// TwinCAT 3 PLC project LabExercise
// ProgramVersion: 3.1.4023.0
// libraries:
//   Tc2_NCI, * (Beckhoff Automation GmbH)
//   Tc2_Standard, * (Beckhoff Automation GmbH)
//   Tc2_System, * (Beckhoff Automation GmbH)
//   Tc3_Module, * (Beckhoff Automation GmbH)
//   VisuDialogs, * (System)
// project tree:
//   Comissioning/Function blocks/ FB_ModifyAutomaticControlSettings.TcPOU (not stored)
//   Comissioning/GVLs/ G_Commissioning.TcGVL (not stored)
//   Comissioning/Struct/ ST_AutomaticControlSettings.TcDUT (not stored), ST_ClosedLoopControlSettings.TcDUT (not stored), ST_MotionReferenceGeneratorSettings.TcDUT (not stored), ST_OpenLoopControlSettings.TcDUT (not stored)
//   ControlBox/Interfaces/ I_ControlBox.TcIO
//   ControlBox/Function blocks/ FB_ControlBox.TcPOU, FB_RealControlBox.TcPOU, FB_VirtualControlBox.TcPOU
//   CraneControl/Function blocks/Sub blocks/ FB_ActiveDamping.TcPOU, FB_Clock.TcPOU, FB_ClosedLoopControl.TcPOU, FB_Joystick.TcPOU, FB_MotionReferenceGenerator_limit.TcPOU, FB_OpenLoopControl.TcPOU, FB_ResetIntegralController.TcPOU, FB_Status.TcPOU
//   CraneControl/Enums/ E_Mode.TcDUT, E_Status.TcDUT
//   CraneControl/Function blocks/Main blocks/ FB_AutomaticControl.TcPOU, FB_ManualControl.TcPOU
//   CraneControl/Functions/ F_BarToEng.TcPOU (not stored), F_LminToEng.TcPOU (not stored), F_RadToDeg.TcPOU (not stored)
//   CraneControl/GVLs/ G_Parameters.TcGVL (not stored), G_Work.TcGVL
//   CraneControl/Struct/ ST_ActiveDamping.TcDUT, ST_Parameters.TcDUT
//   / GlobalTextList.TcGTLO, PlcTask.TcTTO, Simulator.TcTTO (not stored), Visualization Manager.TcVMO (not stored)
//   HMI/ HMI.TcVIS
//   HMI/Sub/ CommissioningHMI.TcVIS, VirtualControlBox.TcVIS
//   Inputs/ FB_JoystickInputScaling.TcPOU, FB_PositionInputScaling.TcPOU, FB_PressureInputScaling.TcPOU, G_Inputs.TcGVL, G_Sensors.TcGVL
//   Inputs/Struct/ ST_AnalogInput.TcDUT (not stored), ST_AnalogInputStatus.TcDUT (not stored)
//   Outputs/ FB_ValveOutput.TcPOU, G_Outputs.TcGVL
//   Outputs/Struct/ ST_pValveDeadBand.TcDUT, ST_ValveOutput.TcDUT
//   ControlBox/GVLs/ G_VirtualControlBox.TcGVL (not stored)
//   Programs/ MAIN.TcPOU, P_Commissioning.TcPOU (not stored), P_ControlBox.TcPOU, P_CraneControl.TcPOU, P_Inputs.TcPOU, P_Outputs.TcPOU, P_Simulator.TcPOU
//   Simulator/ FB_CraneSimulator.TcPOU (not stored), G_Simulator.TcGVL
// real-time tasks:
//   TASK PlcTask: cycle T#1ms, priority 20, ADS port 350
//   TASK Simulator: cycle T#100us, priority 1, ADS port 351
// I/O:
//   DEVICE PLC (EtherCAT), AmsNetId 128.39.203.30.2.1
//     PLC Rack (EK1200) [EK1200-5000 EtherCAT Power supply (2A E-Bus)]
//       DI (EL1008) [EL1008 8Ch. Dig. Input 24V, 3ms]
//       DO (EL2008) [EL2008 8Ch. Dig. Output 24V, 0.5A]
//       End Cap 4 (EL9011) [EL9011 End Terminal]
//   DEVICE RIO (EtherCAT), AmsNetId 128.39.203.30.5.1
//     RIO (EK1100) [EK1100 EtherCAT Coupler (2A E-Bus)]
//       DI (EL1008) [EL1008 8Ch. Dig. Input 24V, 3ms]
//       DO (EL2008) [EL2008 8Ch. Dig. Output 24V, 0.5A]
//       AI1 (EL3068) [EL3068 8Ch. Ana. Input 0-10V]
//       AI2 (EL3068) [EL3068 8Ch. Ana. Input 0-10V]
//       AI3 (EL3174) [EL3174 4Ch. Ana. Input +/-10V Diff., +/-20mA SingleEnded, 16 Bit]
//       AO (EL4104) [EL4104 4Ch. Ana. Output 0-10V, 16bit]
//       End Cap (EL9011) [EL9011 End Terminal]
// variable links:
//   LabExercise/LabExercise Instance <-> PLC (EtherCAT)/PLC Rack (EK1200)/DI (EL1008)
//     PlcTask Inputs/G_Inputs.bTest <-> Channel 1/Input
//   LabExercise/LabExercise Instance <-> PLC (EtherCAT)/PLC Rack (EK1200)/DO (EL2008)
//     PlcTask Outputs/G_Outputs.bTest <-> Channel 1/Output
//   LabExercise/LabExercise Instance <-> RIO (EtherCAT)/RIO (EK1100)/AI1 (EL3068)
//     PlcTask Inputs/G_Inputs.stCylPos.nValue <-> AI Standard Channel 3/Value
//     PlcTask Inputs/G_Inputs.stCylPos.stStatus <-> AI Standard Channel 3/Status
//     PlcTask Inputs/G_Inputs.stJoyX.nValue <-> AI Standard Channel 1/Value
//     PlcTask Inputs/G_Inputs.stJoyX.stStatus <-> AI Standard Channel 1/Status
//     PlcTask Inputs/G_Inputs.stJoyY.nValue <-> AI Standard Channel 2/Value
//     PlcTask Inputs/G_Inputs.stJoyY.stStatus <-> AI Standard Channel 2/Status
//     PlcTask Inputs/G_Inputs.stSpoolPos.nValue <-> AI Standard Channel 4/Value
//     PlcTask Inputs/G_Inputs.stSpoolPos.stStatus <-> AI Standard Channel 4/Status
//   LabExercise/LabExercise Instance <-> RIO (EtherCAT)/RIO (EK1100)/AI2 (EL3068)
//     PlcTask Inputs/G_Inputs.stPressureCompensator.nValue <-> AI Standard Channel 3/Value
//     PlcTask Inputs/G_Inputs.stPressureCompensator.stStatus <-> AI Standard Channel 3/Status
//     PlcTask Inputs/G_Inputs.stPressureLhvSide.nValue <-> AI Standard Channel 5/Value
//     PlcTask Inputs/G_Inputs.stPressureLhvSide.stStatus <-> AI Standard Channel 5/Status
//     PlcTask Inputs/G_Inputs.stPressurePistonSide.nValue <-> AI Standard Channel 4/Value
//     PlcTask Inputs/G_Inputs.stPressurePistonSide.stStatus <-> AI Standard Channel 4/Status
//     PlcTask Inputs/G_Inputs.stPressureReturn.nValue <-> AI Standard Channel 2/Value
//     PlcTask Inputs/G_Inputs.stPressureReturn.stStatus <-> AI Standard Channel 2/Status
//     PlcTask Inputs/G_Inputs.stPressureRodSide.nValue <-> AI Standard Channel 6/Value
//     PlcTask Inputs/G_Inputs.stPressureRodSide.stStatus <-> AI Standard Channel 6/Status
//     PlcTask Inputs/G_Inputs.stPressureSupply.nValue <-> AI Standard Channel 1/Value
//     PlcTask Inputs/G_Inputs.stPressureSupply.stStatus <-> AI Standard Channel 1/Status
//   LabExercise/LabExercise Instance <-> RIO (EtherCAT)/RIO (EK1100)/AI3 (EL3174)
//     PlcTask Inputs/G_Inputs.stFlowReturnSide.nValue <-> AI Standard Channel 1/Value
//     PlcTask Inputs/G_Inputs.stFlowReturnSide.stStatus <-> AI Standard Channel 1/Status
//   LabExercise/LabExercise Instance <-> RIO (EtherCAT)/RIO (EK1100)/AO (EL4104)
//     PlcTask Outputs/G_Outputs.stValveOutput.nValveOutput <-> AO Output Channel 1/Analog output
//   LabExercise/LabExercise Instance <-> RIO (EtherCAT)/RIO (EK1100)/DI (EL1008)
//     PlcTask Inputs/G_Inputs.bAutoModeSelector <-> Channel 1/Input
//     PlcTask Inputs/G_Inputs.bManualModeSelector <-> Channel 2/Input
//     PlcTask Inputs/G_Inputs.bStartButton <-> Channel 3/Input
//     PlcTask Inputs/G_Inputs.bStopButton <-> Channel 4/Input
//   LabExercise/LabExercise Instance <-> RIO (EtherCAT)/RIO (EK1100)/DO (EL2008)
//     PlcTask Outputs/G_Outputs.bGreenLight <-> Channel 1/Output
//     PlcTask Outputs/G_Outputs.bRedLight <-> Channel 2/Output
//     PlcTask Outputs/G_Outputs.stValveOutput.bEnable <-> Channel 3/Output

CONFIGURATION LabExercise
    RESOURCE PLC ON TwinCAT3
        TASK PlcTask(INTERVAL := T#10ms, PRIORITY := 20);
        PROGRAM MAIN WITH PlcTask : MAIN;
    END_RESOURCE
END_CONFIGURATION

// ---- CraneControl/Enums/E_Mode.TcDUT
{attribute 'qualified_only'}
{attribute 'strict'}
TYPE E_Mode :
(
	Off,
	Manual,
	Auto
);
END_TYPE

// ---- CraneControl/Enums/E_Status.TcDUT
{attribute 'qualified_only'}
{attribute 'strict'}
TYPE E_Status :
(
	Off := 0,
	Fault,
	Ready,
	Starting,
	Running,
	Stopping,
	Checking
);
END_TYPE

// ---- CraneControl/Struct/ST_ActiveDamping.TcDUT
TYPE ST_ActiveDamping :
STRUCT
	fFlowGainInverse : LREAL := -1.7153E03;	
	fHPF_Num1 : LREAL := 9.019E-12;
	fHPF_Num2 : LREAL := -9.019E-12;
	fHPF_Den1 : LREAL := 1.0;
	fHPF_Den2 : LREAL := -0.9905;
	fVDI_Num1 : LREAL := 25;
	fVDI_Num2 : LREAL := -48.83;
	fVDI_Num3 : LREAL := 23.85;
	fVDI_Den1 : LREAL := 1;
	fVDI_Den2 : LREAL := -1.721;
	fVDI_Den3 : LREAL := 0.7408;
END_STRUCT
END_TYPE

// ---- CraneControl/Struct/ST_Parameters.TcDUT
TYPE ST_Parameters :
STRUCT
	fCyclicTime 						: LREAL := 0.001; //[s]
	fMaxVelocityLimit 					: LREAL := 0.05; //[m/s]
	stOpenLoopControlSettings 			: ST_OpenLoopControlSettings;
	stClosedLoopControlSettings 		: ST_ClosedLoopControlSettings;
	stPressureFeedback 					: ST_ActiveDamping;
	stValveDeadBand 					: ST_pValveDeadBand;
END_STRUCT
END_TYPE

// ---- Outputs/Struct/ST_pValveDeadBand.TcDUT
TYPE ST_pValveDeadBand :
STRUCT
	fPosMax	: LREAL := 29490; // Positive min value [19660..29490]
	fPosMin	: LREAL := 20889; // Positive max value [19660..29490]
	fNegMin : LREAL := 18441; // Negative max value [9830..19660]
	fNegMax	: LREAL := 9830; // Negative min value [9830..19660]
END_STRUCT
END_TYPE

// ---- Outputs/Struct/ST_ValveOutput.TcDUT
TYPE ST_ValveOutput :
STRUCT
	bEnable					AT %Q* : BOOL := 0;
	nValveOutput 			AT %Q* : INT := 19660;
END_STRUCT
END_TYPE

// ---- CraneControl/GVLs/G_Work.TcGVL
{attribute 'qualified_only'}
VAR_GLOBAL
	eMode 			: E_Mode;
	eStatus 		: E_Status;
	fJoystickY 		: LREAL;
	bFault 			: BOOL;
	bStartButton 	: BOOL;
	bStopButton 	: BOOL;
END_VAR

// ---- Inputs/G_Inputs.TcGVL
{attribute 'qualified_only'}
VAR_GLOBAL
	// PLC Rack
	// Digital Inputs
	bTest 						AT %I* : BOOL;
	
	// RIO Rack
	// Digital Inputs
	bAutoModeSelector			AT %I* : BOOL;
	bManualModeSelector			AT %I* : BOOL;
	bStartButton				AT %I* : BOOL;
	bStopButton					AT %I* : BOOL;
	
	// Analog Inputs 1
	stJoyX 						: ST_AnalogInput;
	stJoyY						: ST_AnalogInput;
	stCylPos 					: ST_AnalogInput;
	stSpoolPos 					: ST_AnalogInput;
	
	// Analog Inputs 2
	stPressureSupply 			: ST_AnalogInput;
	stPressureReturn 			: ST_AnalogInput;
	stPressureCompensator 		: ST_AnalogInput;
	stPressurePistonSide 		: ST_AnalogInput;
	stPressureLhvSide 		    : ST_AnalogInput;
	stPressureRodSide			: ST_AnalogInput;
	
	// Analog Inputs 3 (Multi)
	stFlowReturnSide			: ST_AnalogInput;
END_VAR

// ---- Inputs/G_Sensors.TcGVL
{attribute 'qualified_only'}
VAR_GLOBAL
	fJoystickY 			: LREAL;
	fPistonPosition 	: LREAL;
	fPressureSupply		: LREAL;
	fPressureReturn 	: LREAL;
	fPressurePistonSide : LREAL;
	fPressureLhvSide  	: LREAL;
	fPressureRodSide 	: LREAL;
END_VAR

// ---- Outputs/G_Outputs.TcGVL
{attribute 'qualified_only'}
VAR_GLOBAL
	// PLC Rack
	// Digital Outputs
	bTest					 AT %Q* : BOOL;
	
	// RIO Rack
	// Digital Outputs
	bGreenLight 			AT %Q* : BOOL;
	bRedLight 				AT %Q* : BOOL;
	// Analog Outputs
	stValveOutput : ST_ValveOutput;
END_VAR

// ---- Simulator/G_Simulator.TcGVL
{attribute 'qualified_only'}
VAR_GLOBAL
	bSimulatorOn : BOOL;
	fPistonSidePressure : LREAL;
	fRodSidePressure 	: LREAL;
	fPistonPosition 	: LREAL;
END_VAR

// ---- ControlBox/Interfaces/I_ControlBox.TcIO
INTERFACE I_ControlBox

METHOD Lamps 
VAR_INPUT
	bEnable : BOOL;
END_VAR
END_METHOD

METHOD ModeSelector 
VAR_INPUT
END_VAR
VAR_OUTPUT
	eMode : E_Mode;
END_VAR
END_METHOD

END_INTERFACE

// ---- Programs/MAIN.TcPOU
PROGRAM MAIN
VAR
END_VAR

P_Commissioning();
P_ControlBox();
P_CraneControl();
P_Outputs();
P_Inputs();

END_PROGRAM

// ---- Programs/P_ControlBox.TcPOU
PROGRAM P_ControlBox
VAR
	fbControlBox : FB_ControlBox; 
END_VAR

fbControlBox(
bRealControlBox := TRUE,
eStatus := G_Work.eStatus,
eMode => G_Work.eMode,
);

END_PROGRAM

// ---- ControlBox/Function blocks/FB_ControlBox.TcPOU
FUNCTION_BLOCK FB_ControlBox
VAR_INPUT
	bRealControlBox : BOOL;
	eStatus : E_Status;
END_VAR
VAR_OUTPUT
	eMode : E_Mode;
END_VAR
VAR
	fbVirtualControlBox : FB_VirtualControlBox;
	fbRealControlBox : FB_RealControlBox;
	fbSelectedControlBox : I_ControlBox := fbVirtualControlBox;
END_VAR

IF bRealControlBox THEN
	fbSelectedControlBox := fbRealControlBox;
ELSE
	fbSelectedControlBox := fbVirtualControlBox;
END_IF	
	
fbSelectedControlBox.ModeSelector(
	eMode => eMode
);

fbSelectedControlBox.PushButtons(
	eMode := eMode,
	eStatus := eStatus,
	bStart => G_Work.bStartButton,
	bStop => G_Work.bStopButton 	
);

fbSelectedControlBox.Lamps(
	eMode := eMode,
	eStatus := eStatus
);

fbSelectedControlBox.Joystick(
	eMode := eMode,
	eStatus := eStatus,
	fJoystickY => G_Work.fJoystickY
);

END_FUNCTION_BLOCK

// ---- ControlBox/Function blocks/FB_VirtualControlBox.TcPOU
FUNCTION_BLOCK FB_VirtualControlBox IMPLEMENTS I_ControlBox
VAR_INPUT
END_VAR
VAR_OUTPUT
END_VAR
VAR
END_VAR

METHOD Lamps
VAR_INPUT
	bEnable : BOOL;
END_VAR
IF bEnable THEN 
	IF G_Work.eStatus = E_Status.Running THEN
		G_VirtualControlBox.bGreenLight :=  TRUE;
	ELSE
		G_VirtualControlBox.bGreenLight :=  FALSE;
	END_IF
	
	IF G_Work.eStatus = E_Status.Fault THEN
		G_VirtualControlBox.bRedLight :=  TRUE;
	ELSE
		G_VirtualControlBox.bRedLight :=  FALSE;
	END_IF
END_IF
END_METHOD

METHOD ModeSelector 
VAR_INPUT
END_VAR
VAR_OUTPUT
	eMode : E_Mode;
END_VAR
CASE eMode OF 
	E_Mode.Off:	
		IF G_VirtualControlBox.bOnSelector AND NOT(G_VirtualControlBox.bAutoSelector) THEN	
			eMode := E_Mode.Manual;
		END_IF
		
		IF G_VirtualControlBox.bOnSelector AND G_VirtualControlBox.bAutoSelector THEN	
			eMode := E_Mode.Auto;
		END_IF

	E_Mode.Manual: 
		IF NOT(G_VirtualControlBox.bOnSelector) THEN	
			eMode := E_Mode.Off;
		END_IF
		
		IF G_VirtualControlBox.bOnSelector AND G_VirtualControlBox.bAutoSelector THEN	
			eMode := E_Mode.Auto;
		END_IF
	
	E_Mode.Auto:
		IF NOT(G_VirtualControlBox.bOnSelector) THEN	
			eMode := E_Mode.Off;
		END_IF
		
		IF G_VirtualControlBox.bOnSelector AND NOT(G_VirtualControlBox.bAutoSelector) THEN	
			eMode := E_Mode.Manual;
		END_IF	
ELSE 	
	eMode := E_Mode.Off;
END_CASE
END_METHOD

END_FUNCTION_BLOCK

// ---- ControlBox/Function blocks/FB_RealControlBox.TcPOU
FUNCTION_BLOCK FB_RealControlBox IMPLEMENTS I_ControlBox
VAR_INPUT
END_VAR
VAR_OUTPUT
END_VAR
VAR
END_VAR

METHOD Joystick
VAR_INPUT
	eMode 	: E_Mode;
	eStatus : E_Status;
END_VAR
VAR_OUTPUT
	fJoystickY : LREAL;
END_VAR
IF eMode = E_Mode.Manual AND eStatus = E_Status.Running THEN
	fJoystickY := G_Sensors.fJoystickY;
ELSE
	fJoystickY := 0.0;
END_IF
END_METHOD

METHOD Lamps 
VAR_INPUT
	eMode 	: E_Mode;
	eStatus : E_Status;
END_VAR
IF eStatus = E_Status.Running AND NOT(eMode = E_Mode.Off) THEN
	G_Outputs.bGreenLight :=  TRUE;
ELSE
	G_Outputs.bGreenLight :=  FALSE;
END_IF

IF eStatus = E_Status.Fault  AND NOT(eMode = E_Mode.Off) THEN
	G_Outputs.bRedLight :=  TRUE;
ELSE
	G_Outputs.bRedLight :=  FALSE;
END_IF
END_METHOD

METHOD ModeSelector 
VAR_INPUT
END_VAR
VAR_OUTPUT
	eMode : E_Mode;
END_VAR
CASE eMode OF 
	E_Mode.Off:	
		IF G_Inputs.bManualModeSelector AND NOT(G_Inputs.bAutoModeSelector) THEN	
			eMode := E_Mode.Manual;
		END_IF
		
		IF G_Inputs.bAutoModeSelector AND NOT(G_Inputs.bManualModeSelector) THEN	
			eMode := E_Mode.Auto;
		END_IF

	E_Mode.Manual: 
		IF NOT(G_Inputs.bManualModeSelector) AND NOT(G_Inputs.bManualModeSelector) THEN	
			eMode := E_Mode.Off;
		END_IF
		
		IF G_Inputs.bAutoModeSelector AND NOT(G_Inputs.bManualModeSelector) THEN	
			eMode := E_Mode.Auto;
		END_IF
	
	E_Mode.Auto:
		IF NOT(G_Inputs.bManualModeSelector) AND NOT(G_Inputs.bManualModeSelector) THEN	
			eMode := E_Mode.Off;
		END_IF
		
		IF G_Inputs.bManualModeSelector AND NOT(G_Inputs.bAutoModeSelector) THEN	
			eMode := E_Mode.Manual;
		END_IF	
ELSE 	
	eMode := E_Mode.Off;
END_CASE
END_METHOD

METHOD PushButtons
VAR_INPUT
	eMode 	: E_Mode;
	eStatus : E_Status;
END_VAR
VAR_OUTPUT
	bStart : BOOL;
	bStop : BOOL;
END_VAR
IF NOT(eMode = E_Mode.Off) AND (NOT(eStatus = E_Status.Fault) OR (eStatus = E_Status.Off)) THEN 
	bStart := G_Inputs.bStartButton;
	bStop := G_Inputs.bStopButton;
ELSE
	bStart := FALSE;
	bStop := FALSE;
END_IF
END_METHOD

END_FUNCTION_BLOCK

// ---- Programs/P_CraneControl.TcPOU
PROGRAM P_CraneControl
VAR
 	fbStatus 					: FB_Status;
	fbRunningClock 				: FB_Clock;
	fbManualControl 			: FB_ManualControl; 
	bEnableManualControl 		: BOOL;
	fbAutomaticControl 			: FB_AutomaticControl;
	bEnableAutomaticControl 	: BOOL; 
	fbActiveDamping 			: FB_ActiveDamping;
	fControlOutputNormalized 	: LREAL; 
	
	ADtest0 : LREAL;
	ADtest1 : LREAL;
	ADtest2 : LREAL;
	ADtest : BOOL;
END_VAR

fbStatus(
bFault := G_Work.bFault,
eMode := G_Work.eMode,
fTime := fbRunningClock.fTime,
eStatus => G_Work.eStatus
);

fbRunningClock(
	bStart := (fbStatus.eStatus = E_Status.Starting) OR (fbStatus.eStatus = E_Status.Running),
	bStop := (fbStatus.eStatus = E_Status.Stopping),
	fCycleTime := G_Parameters.stParam.fCyclicTime
);

fbManualControl(
	eMode := G_Work.eMode,
	eStatus := G_Work.eStatus,
	stParam := G_Parameters.stParam, 
);

fbAutomaticControl(
	eMode := G_Work.eMode,
	eStatus := G_Work.eStatus,
	stAutomaticControlSettings := G_Commissioning.stAutomaticControlSettings,
	stMotionReferenceGeneratorSettings := G_Commissioning.stMotionReferenceGeneratorSettings,
	stParam := G_Parameters.stParam,
	fPositionFeedback := G_Sensors.fPistonPosition
);

fbActiveDamping(
	ssMethodType := BOOL_TO_SINT(G_Commissioning.stAutomaticControlSettings.bEnableActiveDamping),
	bEnable := (fbStatus.eStatus = E_Status.Running),
	stParam := G_Parameters.stParam,
	fPressurePistonSide_Pa := F_BarToEng(G_Sensors.fPressurePistonSide),
	fPressureRodSide_Pa := F_BarToEng(G_Sensors.fPressureRodSide)
);

IF (G_Work.eMode = E_Mode.Manual AND G_Work.eStatus = E_Status.Running) THEN
	fControlOutputNormalized := LIMIT(-1.0, (fbManualControl.fControlOutputNormalized - fbActiveDamping.fPressureFeedbackNormalized), 1.0);
ELSIF (G_Work.eMode = E_Mode.Auto AND G_Work.eStatus = E_Status.Running) THEN
	fControlOutputNormalized := LIMIT(-1.0, (-fbAutomaticControl.fControlOutputNormalized - fbActiveDamping.fPressureFeedbackNormalized), 1.0);
ELSE
	fControlOutputNormalized := 0.0;
END_IF

G_Work.fControlOutputNormalized := fControlOutputNormalized;

END_PROGRAM

// ---- CraneControl/Function blocks/Sub blocks/FB_Status.TcPOU
FUNCTION_BLOCK FB_Status
VAR_INPUT
	eMode 	: E_Mode;
	fTime	: LREAL;
	bFault 	: BOOL;
END_VAR
VAR_OUTPUT
	eStatus : E_Status := E_Status.Checking;
END_VAR
VAR
	bRunning : BOOL;
END_VAR

IF fTime > 2.0 THEN
	bRunning := TRUE;
ELSE
	bRunning := FALSE;	
END_IF


CASE eStatus OF 
	E_Status.Checking:
		IF bFault THEN
			eStatus := E_Status.Fault;
		END_IF
		
		IF NOT(eMode = E_Mode.Off) AND NOT(bFault)THEN	
			eStatus := E_Status.Ready;
		END_IF
		
		IF eMode = E_Mode.Off THEN	
			eStatus := E_Status.Off;
		END_IF
		
	E_Status.Off:	
		IF NOT(eMode = E_Mode.Off) THEN	
			eStatus := E_Status.Checking;
		END_IF

	E_Status.Fault:
		IF NOT(bFault) THEN
			eStatus := E_Status.Checking;
		END_IF
	
	E_Status.Ready:
		IF G_Work.bStartButton AND NOT(eMode = E_Mode.Off) AND NOT(bFault) THEN
			eStatus := E_Status.Starting;
		END_IF	
		
		IF  eMode = E_Mode.Off OR bFault THEN
			eStatus := E_Status.Checking;
		END_IF	

	E_Status.Starting:
		IF bRunning THEN
			eStatus := E_Status.Running;
		END_IF 
		
		IF bFault OR eMode = E_Mode.Off  THEN
			eStatus := E_Status.Checking;
		END_IF
		
	
	E_Status.Running:
	
		IF G_Work.bStopButton THEN
			eStatus := E_Status.Stopping;
		END_IF
		
		IF NOT(bRunning) OR eMode = E_Mode.Off OR bFault THEN
			eStatus := E_Status.Checking;
		END_IF
	
	E_Status.Stopping:	
		IF NOT(bRunning) THEN
			eStatus := E_Status.Checking;
		END_IF
	
		IF eMode = E_Mode.Off OR bFault THEN
		eStatus := E_Status.Checking;
		END_IF	
	
ELSE 	
	eStatus := E_Status.Checking;
END_CASE

END_FUNCTION_BLOCK

// ---- CraneControl/Function blocks/Sub blocks/FB_Clock.TcPOU
FUNCTION_BLOCK FB_Clock
VAR_INPUT
	bStart : BOOL;
	bStop : BOOL;
	fCycleTime : LREAL;
END_VAR
VAR_OUTPUT
	fTime : LREAL;
END_VAR
VAR
END_VAR

IF bStart AND NOT(bStop) THEN
	fTime := fTime + fCycleTime;
ELSE
	fTime := 0.0;
END_IF

END_FUNCTION_BLOCK

// ---- CraneControl/Function blocks/Main blocks/FB_ManualControl.TcPOU
FUNCTION_BLOCK FB_ManualControl
VAR_INPUT
	eMode : E_Mode;
	eStatus : E_Status;
	stParam : ST_Parameters;
END_VAR
VAR_OUTPUT
	fVelocityFeedForwardControlOutput : LREAL;
END_VAR
VAR
	fbJoystick : FB_Joystick; 
	fbOpenLoopControl : FB_OpenLoopControl; 
END_VAR

fbJoystick(
	bEnable := (eMode = E_Mode.Manual),
	stParam := stParam,
	fNormalizedInput := Work.fJoystickY,
);

fbOpenLoopControl(
	bEnable := (eMode = E_Mode.Manual),
	stParam := stParam,
	fInput_ms := fbJoystick.fOuput,
	fNormalizedOutput => fVelocityFeedForwardControlOutput
);

END_FUNCTION_BLOCK

// ---- CraneControl/Function blocks/Sub blocks/FB_Joystick.TcPOU
FUNCTION_BLOCK FB_Joystick
VAR_INPUT
	bEnable : BOOL;
	fNormalizedInput : LREAL;
	stParam : ST_Parameters;
END_VAR
VAR_OUTPUT
	fOuput : LREAL;
END_VAR
VAR
END_VAR

IF bEnable THEN
	fOuput := fNormalizedInput*Parameters.stParam.fMaxVelocityLimit;
ELSE
	fOuput := 0.0;
END_IF

END_FUNCTION_BLOCK

// ---- CraneControl/Function blocks/Sub blocks/FB_OpenLoopControl.TcPOU
FUNCTION_BLOCK FB_OpenLoopControl
VAR_INPUT
	bEnable: BOOL;
	fInput_ms: LREAL;
	stParam : ST_Parameters;
END_VAR
VAR_OUTPUT
	fNormalizedOutput: LREAL;
END_VAR
VAR
	fFlowReference_m3s : LREAL;
	fM3sToLmin : LREAL := 60000;
END_VAR

IF fInput_ms >= 0.0 THEN 
    fFlowReference_m3s := stparam.stOpenLoopControl.fBoreArea * fInput_ms;
ELSE 
    fFlowReference_m3s := fInput_ms * stparam.stOpenLoopControl.fAnnulusArea;
END_IF;

IF bEnable THEN 
    fNormalizedOutput := (fM3sToLmin * fFlowReference_m3s) / stParam.stOpenLoopControl.fMaxFlowCapacity;
ELSE 
    fNormalizedOutput := 0.0;
END_IF;

IF fNormalizedOutput > 1.0 THEN 
    fNormalizedOutput := 1.0;
ELSIF fNormalizedOutput < -1.0 THEN 
    fNormalizedOutput := -1.0;
END_IF;

END_FUNCTION_BLOCK

// ---- CraneControl/Function blocks/Main blocks/FB_AutomaticControl.TcPOU
FUNCTION_BLOCK FB_AutomaticControl
VAR_INPUT
	eMode 								: E_Mode;
	eStatus 							: E_Status;
	bStopMotion 						: BOOL;
	stMotionReferenceGeneratorSettings  : ST_MotionReferenceGeneratorSettings;
	stAutomaticControlSettings 			: ST_AutomaticControlSettings;
	stParam 							: ST_Parameters; 
	fPositionFeedback					: LREAL;
END_VAR
VAR_OUTPUT
	fTime : LREAL;
	fControlOutputNormalized : LREAL;
END_VAR
VAR
	fbClock : FB_Clock;	
	fbMotionReferenceGenerator 		: FB_MotionReferenceGenerator_limit;	
	fbVelocityFeedForwardControl 	: FB_OpenLoopControl;
	fbResetIntegralController 		: FB_ResetIntegralController; 
	fbClosedLoopPositionControl 	: FB_ClosedLoopControl;
END_VAR

fbClock(
	bStart := (eMode = E_Mode.Auto AND (eStatus = E_Status.Starting OR eStatus = E_Status.Running)),
	bStop := bStopMotion,
	fCycleTime := stParam.fCyclicTime
);

fbMotionReferenceGenerator(
	bEnable := (eMode = E_Mode.Auto AND eStatus = E_Status.Running),
	stMotionReferenceGeneratorSettings := stMotionReferenceGeneratorSettings,
	fClock_s := fbClock.fTime
);

fbVelocityFeedForwardControl(
	bEnable := stAutomaticControlSettings.bEnableVelocityFeedForwardControl,
	stParam := stParam,
	fInput_ms := fbMotionReferenceGenerator.fVelocityReference_ms
);

fbResetIntegralController(
	stParam := stParam,
	fPositionError_m := fbClosedLoopPositionControl.fPositionError,
	fVelocityReference_ms := fbMotionReferenceGenerator.fVelocityReference_ms
);

fbClosedLoopPositionControl(
	bEnable := stAutomaticControlSettings.bEnableClosedLoopPositionControl,
	stParam := stParam,
	bActivateIntegralController := stAutomaticControlSettings.bEnableIntegralController,
	bIntegralControllReset := fbResetIntegralController.bReset,
	fInput_m := fbMotionReferenceGenerator.fPositionReference_m,
	fFeedback_m := fPositionFeedback
);

IF (eMode = E_Mode.Auto AND eStatus = E_Status.Running) THEN
	fControlOutputNormalized := LIMIT(-1.0, (fbVelocityFeedForwardControl.fNormalizedOutput + fbClosedLoopPositionControl.fNormalizedOutput), 1.0);
ELSE
	fControlOutputNormalized := 0.0;
END_IF

END_FUNCTION_BLOCK

// ---- CraneControl/Function blocks/Sub blocks/FB_MotionReferenceGenerator_limit.TcPOU
FUNCTION_BLOCK FB_MotionReferenceGenerator_limit
VAR_INPUT
	bEnable 							: BOOL;
	stMotionReferenceGeneratorSettings  : ST_MotionReferenceGeneratorSettings;
	fClock_s							: LREAL;
END_VAR
VAR_OUTPUT
	fPositionReference_m	: LREAL;
	fVelocityReference_ms	: LREAL;
	fTotalMotionTime_s		: LREAL;
	bErrorSignal			: BOOL;
END_VAR
VAR
	fStartPosition_m		: LREAL;
	fStartVelocity_m		: LREAL;
	fPositionSetpoint_ms	: LREAL;
	fVelocitySetpoint_m		: LREAL;
	fTimeBeforeStarting_s	: LREAL;
	fRampTime_s				: LREAL;
	fHoldPositionTime_s		: LREAL;
	Error					: DINT;
	slopeExt				: LREAL;
	slopeRetr				: LREAL;
	tHold					: LREAL;
	x1						: LREAL;
	x4						: LREAL;
	x1_tmp					: LREAL;
	x1_tmp_tmp				: LREAL;
	x4_tmp					: LREAL;
	x4_tmp_tmp				: LREAL;
	x4_tmp_tmp_0			: LREAL;
	x1_tmp_0				: LREAL;
END_VAR

IF NOT(bEnable) THEN
	RETURN;
END_IF

// LIMIT function: https://help.codesys.com/api-content/2/codesys/3.5.12.0/en/_cds_operator_limit/
fStartPosition_m := LIMIT(stMotionReferenceGeneratorSettings.fMinPosition, stMotionReferenceGeneratorSettings.fStartPosition_m, stMotionReferenceGeneratorSettings.fMaxPosition);
fStartVelocity_m := LIMIT(0.0, stMotionReferenceGeneratorSettings.fStartVelocity_m, stMotionReferenceGeneratorSettings.fMaxVelocity);
fPositionSetpoint_ms := LIMIT(stMotionReferenceGeneratorSettings.fMinPosition, stMotionReferenceGeneratorSettings.fPositionSetpoint_ms, stMotionReferenceGeneratorSettings.fMaxPosition);
fVelocitySetpoint_m := LIMIT(0.0, stMotionReferenceGeneratorSettings.fVelocitySetpoint_m, stMotionReferenceGeneratorSettings.fMaxVelocity);
fTimeBeforeStarting_s := LIMIT(0.0, stMotionReferenceGeneratorSettings.fTimeBeforeStarting_s, 10.0);
fRampTime_s := LIMIT(0.0, stMotionReferenceGeneratorSettings.fRampTime_s, 10.0);
fHoldPositionTime_s := LIMIT(0.0, stMotionReferenceGeneratorSettings.fHoldPositionTime_s, 60.0);

slopeExt := fStartVelocity_m - fVelocitySetpoint_m;

slopeRetr := ( -fVelocitySetpoint_m) - fStartVelocity_m;

tHold := ((fPositionSetpoint_ms - fStartPosition_m) - (((fVelocitySetpoint_m * fVelocitySetpoint_m) - (fStartVelocity_m * fStartVelocity_m)) / (fVelocitySetpoint_m / fRampTime_s))) / fVelocitySetpoint_m;

IF tHold < 0.0  THEN 
    bErrorSignal := TRUE;
ELSE 
    bErrorSignal := FALSE;
END_IF;

x1_tmp_tmp := fTimeBeforeStarting_s + fRampTime_s;
x1_tmp := x1_tmp_tmp - fTimeBeforeStarting_s;
x1_tmp_0 := slopeExt / fRampTime_s;
x1 := ((x1_tmp * fStartVelocity_m) + fStartPosition_m) - ((x1_tmp_0 * (x1_tmp * x1_tmp)) / 2.0);

x4_tmp_tmp := x1_tmp_tmp + tHold;
x4_tmp_tmp_0 := x4_tmp_tmp + fRampTime_s;
x4_tmp := x4_tmp_tmp_0 + fHoldPositionTime_s;
x1_tmp := x4_tmp + fRampTime_s;
x4 := x1_tmp - x4_tmp;
x4 := (fPositionSetpoint_ms - (x4 * fStartVelocity_m)) + (((slopeRetr / fRampTime_s) * (x4 * x4)) / 2.0);

IF Error = 1 THEN 
    fPositionReference_m := fStartPosition_m;
    fVelocityReference_ms := fStartVelocity_m;
ELSIF (fClock_s >= 0.0) AND (fClock_s < fTimeBeforeStarting_s) THEN 
    fPositionReference_m := fStartPosition_m;
    fVelocityReference_ms := fStartVelocity_m;
ELSIF (fClock_s >= fTimeBeforeStarting_s) AND (fClock_s < x1_tmp_tmp) THEN 
    slopeRetr := fClock_s - fTimeBeforeStarting_s;
    fPositionReference_m := ((slopeRetr * fStartVelocity_m) + fStartPosition_m) - ((x1_tmp_0 * (slopeRetr * slopeRetr)) / 2.0);
    fVelocityReference_ms := fStartVelocity_m - (x1_tmp_0 * slopeRetr);
ELSIF (fClock_s >= x1_tmp_tmp) AND (fClock_s < x4_tmp_tmp) THEN 
    fPositionReference_m := ((fClock_s - x1_tmp_tmp) * fVelocitySetpoint_m) + x1;
    fVelocityReference_ms := fVelocitySetpoint_m;
ELSIF (fClock_s >= x4_tmp_tmp) AND (fClock_s < x4_tmp_tmp_0) THEN 
    slopeRetr := fClock_s - x4_tmp_tmp;
    fPositionReference_m := ((((x4_tmp_tmp - x1_tmp_tmp) * fVelocitySetpoint_m) + x1) + (slopeRetr * fVelocitySetpoint_m)) + ((x1_tmp_0 * (slopeRetr * slopeRetr)) / 2.0);
    fVelocityReference_ms := (slopeRetr * (slopeExt / fRampTime_s)) + fVelocitySetpoint_m;
ELSIF (fClock_s >= x4_tmp_tmp_0) AND (fClock_s < x4_tmp) THEN 
    fPositionReference_m := fPositionSetpoint_ms;
    fVelocityReference_ms := fStartVelocity_m;
ELSIF (fClock_s >= x4_tmp) AND (fClock_s < x1_tmp) THEN 
    slopeExt := fClock_s - x4_tmp;
    slopeRetr := slopeRetr / fRampTime_s;
    fPositionReference_m := (fPositionSetpoint_ms - (slopeExt * fStartVelocity_m)) + ((slopeRetr * (slopeExt * slopeExt)) / 2.0);
    fVelocityReference_ms := (slopeExt * slopeRetr) + fStartVelocity_m;
ELSE 
    x1_tmp_0 := x1_tmp + tHold;

    IF (fClock_s >= x1_tmp) AND (fClock_s < x1_tmp_0) THEN 
        fPositionReference_m := x4 - ((fClock_s - x1_tmp) * fVelocitySetpoint_m);
        fVelocityReference_ms :=  -fVelocitySetpoint_m;
    ELSIF (fClock_s >= x1_tmp_0) AND (fClock_s < (((((((fTimeBeforeStarting_s + fRampTime_s) + tHold) + fRampTime_s) + fHoldPositionTime_s) + fRampTime_s) + tHold) + fRampTime_s)) THEN 
        slopeExt := fClock_s - x1_tmp_0;
        slopeRetr := slopeRetr / fRampTime_s;
        fPositionReference_m := ((x4 - ((x1_tmp_0 - x1_tmp) * fVelocitySetpoint_m)) - (slopeExt * fVelocitySetpoint_m)) - ((slopeRetr * (slopeExt * slopeExt)) / 2.0);
        fVelocityReference_ms := ( -fVelocitySetpoint_m) - (slopeExt * slopeRetr);
    ELSE 
        fPositionReference_m := fStartPosition_m;
        fVelocityReference_ms := fStartVelocity_m;
    END_IF;

END_IF;

fTotalMotionTime_s := ((((((fTimeBeforeStarting_s + fRampTime_s) + tHold) + fRampTime_s) + fHoldPositionTime_s) + fRampTime_s) + tHold) + fRampTime_s;

END_FUNCTION_BLOCK

// ---- CraneControl/Function blocks/Sub blocks/FB_ResetIntegralController.TcPOU
FUNCTION_BLOCK FB_ResetIntegralController
VAR_INPUT
	stParam : ST_Parameters;
	fVelocityReference_ms: LREAL;
	fPositionError_m: LREAL;
END_VAR
VAR_OUTPUT
	bReset: BOOL;
END_VAR
VAR
END_VAR

IF ABS(fVelocityReference_ms) > 0.0 THEN 
    bReset := FALSE;
ELSIF ABS(fPositionError_m) > stParam.stClosedLoopControl.fMaxPositionError THEN 
    bReset := FALSE;
ELSE 
    bReset := TRUE;
END_IF;

END_FUNCTION_BLOCK

// ---- CraneControl/Function blocks/Sub blocks/FB_ClosedLoopControl.TcPOU
FUNCTION_BLOCK FB_ClosedLoopControl
VAR_INPUT
	bEnable: BOOL;
	stParam : ST_Parameters;
	bActivateIntegralController: BOOL;
	bIntegralControllReset: BOOL;
	fInput_m: LREAL;
	fFeedback_m: LREAL;
END_VAR
VAR_OUTPUT
	fNormalizedOutput: LREAL;
	fPositionError: LREAL;
END_VAR
VAR
	rtb_u_FB: LREAL;
	rtb_Saturation1: LREAL;
	c_DiscreteTimeIntegrator_DS: LREAL;
END_VAR

fPositionError := fInput_m - fFeedback_m;

IF bIntegralControllReset THEN 
	c_DiscreteTimeIntegrator_DS := 0.0;
END_IF;

IF c_DiscreteTimeIntegrator_DS >= 1.0 THEN 
	c_DiscreteTimeIntegrator_DS := 1.0;
ELSIF c_DiscreteTimeIntegrator_DS <= -1.0 THEN 
	c_DiscreteTimeIntegrator_DS := -1.0;
END_IF;

IF bActivateIntegralController THEN 
	rtb_u_FB := c_DiscreteTimeIntegrator_DS;
ELSE 
	rtb_u_FB := 0.0;
END_IF;

rtb_u_FB := (stParam.stClosedLoopControl.fProportionalGain * fPositionError) + rtb_u_FB;

IF rtb_u_FB > 1.0 THEN 
	rtb_Saturation1 := 1.0;
ELSIF rtb_u_FB >= -1.0 THEN 
	rtb_Saturation1 := rtb_u_FB;
ELSE 
	rtb_Saturation1 := -1.0;
END_IF;

IF bEnable THEN 
	fNormalizedOutput := rtb_Saturation1;
ELSE 
	fNormalizedOutput := 0.0;
END_IF;

c_DiscreteTimeIntegrator_DS := (((((rtb_Saturation1 - rtb_u_FB) / stParam.stClosedLoopControl.fProportionalGain) + fPositionError) * stParam.stClosedLoopControl.fIntegralGain) * stParam.fCyclicTime) + c_DiscreteTimeIntegrator_DS;

IF c_DiscreteTimeIntegrator_DS >= 1.0 THEN 
	c_DiscreteTimeIntegrator_DS := 1.0;
ELSIF c_DiscreteTimeIntegrator_DS <= -1.0 THEN 
	c_DiscreteTimeIntegrator_DS := -1.0;
END_IF;

END_FUNCTION_BLOCK

// ---- CraneControl/Function blocks/Sub blocks/FB_ActiveDamping.TcPOU
FUNCTION_BLOCK FB_ActiveDamping
VAR_INPUT
	ssMethodType: SINT;
	bEnable: BOOL;
	stParam : ST_Parameters;
	fPressurePistonSide_Pa	: LREAL;
	fPressureRodSide_Pa		: LREAL;
END_VAR
VAR_OUTPUT
	fPressureFeedbackNormalized: LREAL;
END_VAR
VAR
	rtb_Switch3: LREAL;
	HighPassFilter_tmp: LREAL;
	VectorConcatenate: ARRAY[0..1] OF LREAL;
	VectorConcatenate1: ARRAY[0..1] OF LREAL;
	VectorConcatenate2: ARRAY[0..2] OF LREAL;
	VectorConcatenate3: ARRAY[0..2] OF LREAL;
	HighPassFilter_states: LREAL;
	ValveDynamicsInverse_states: ARRAY[0..1] OF LREAL;
END_VAR

CASE ssMethodType OF
    0: 
        HighPassFilter_states := 0.0;
        ValveDynamicsInverse_states[0] := 0.0;
        ValveDynamicsInverse_states[1] := 0.0;

    1: 
        IF bEnable THEN 
            rtb_Switch3 := 0.0;
        ELSE 
            rtb_Switch3 := 1.0;
        END_IF;

        VectorConcatenate[0] := stParam.stPressureFeedback.fHPF_Num1;
        VectorConcatenate[1] := stParam.stPressureFeedback.fHPF_Num2;
        VectorConcatenate1[0] := stParam.stPressureFeedback.fHPF_Den1;
        VectorConcatenate1[1] := stParam.stPressureFeedback.fHPF_Den2;
        VectorConcatenate2[0] := stParam.stPressureFeedback.fVDI_Num1;
        VectorConcatenate2[1] := stParam.stPressureFeedback.fVDI_Num2;
        VectorConcatenate2[2] := stParam.stPressureFeedback.fVDI_Num3;
        VectorConcatenate3[0] := stParam.stPressureFeedback.fVDI_Den1;
        VectorConcatenate3[1] := stParam.stPressureFeedback.fVDI_Den2;
        VectorConcatenate3[2] := stParam.stPressureFeedback.fVDI_Den3;

        IF rtb_Switch3 <> 0.0 THEN 
            HighPassFilter_states := 0.0;
        END_IF;

        HighPassFilter_tmp := (fPressurePistonSide_Pa*1.4083 - (fPressureRodSide_Pa)) - (VectorConcatenate1[1] * HighPassFilter_states);
		
        fPressureFeedbackNormalized := ((VectorConcatenate[0] * HighPassFilter_tmp) + (VectorConcatenate[1] * HighPassFilter_states)) * stParam.stPressureFeedback.fFlowGainInverse;

        IF fPressureFeedbackNormalized > 1.0 THEN 
            fPressureFeedbackNormalized := 1.0;
        ELSIF fPressureFeedbackNormalized < -1.0 THEN 
            fPressureFeedbackNormalized := -1.0;
        END_IF;

        IF rtb_Switch3 <> 0.0 THEN 
            ValveDynamicsInverse_states[0] := 0.0;
            ValveDynamicsInverse_states[1] := 0.0;
        END_IF;

        rtb_Switch3 := (fPressureFeedbackNormalized - (ValveDynamicsInverse_states[0] * VectorConcatenate3[1])) - (ValveDynamicsInverse_states[1] * VectorConcatenate3[2]);

        IF bEnable THEN 
            fPressureFeedbackNormalized := ((VectorConcatenate2[0] * rtb_Switch3) + (ValveDynamicsInverse_states[0] * VectorConcatenate2[1])) + (ValveDynamicsInverse_states[1] * VectorConcatenate2[2]);
        ELSE 
            fPressureFeedbackNormalized := 0.0;
        END_IF;

        IF fPressureFeedbackNormalized > 1.0 THEN 
            fPressureFeedbackNormalized := 1.0;
        ELSIF fPressureFeedbackNormalized < -1.0 THEN 
            fPressureFeedbackNormalized := -1.0;
        END_IF;

        HighPassFilter_states := HighPassFilter_tmp;

        ValveDynamicsInverse_states[1] := ValveDynamicsInverse_states[0];
        ValveDynamicsInverse_states[0] := rtb_Switch3;
END_CASE;

END_FUNCTION_BLOCK

// ---- Programs/P_Outputs.TcPOU
PROGRAM P_Outputs
VAR
	stValveOutput : FB_ValveOutput;
END_VAR

stValveOutput(
	bEnable := (G_Work.eStatus = E_Status.Running),
	stParam := G_Parameters.stParam,
	fNormalizedInput := G_Work.fControlOutputNormalized,
	bEnableValveOutput => G_Outputs.stValveOutput.bEnable,
	nOutput => G_Outputs.stValveOutput.nValveOutput
);

END_PROGRAM

// ---- Outputs/FB_ValveOutput.TcPOU
FUNCTION_BLOCK FB_ValveOutput
VAR_INPUT
	bEnable 			: BOOL;
	stParam 			: ST_Parameters;
	fNormalizedInput 	: LREAL;
END_VAR
VAR_OUTPUT
	bEnableValveOutput : BOOL;
	nOutput : INT; 
END_VAR
VAR
	nOffset 	: INT := 19660;
	nMaxValue	: INT := 29490;
	nMinValue 	: INT :=  9830;
	nTempOutput : INT;
END_VAR

IF fNormalizedInput > 0.0 THEN
	nTempOutput := LREAL_TO_INT(ABS(fNormalizedInput*(stParam.stValveDeadBand.fPosMax - stParam.stValveDeadBand.fPosMin) + stParam.stValveDeadBand.fPosMin));
ELSIF fNormalizedInput < 0.0 THEN
	nTempOutput := LREAL_TO_INT(ABS(fNormalizedInput*(stParam.stValveDeadBand.fNegMax - stParam.stValveDeadBand.fNegMin) - stParam.stValveDeadBand.fNegMin));
ELSE
	nTempOutput := nOffset;
END_IF

IF NOT(bEnable) THEN
	nOutput := nOffset;
	bEnableValveOutput := FALSE;
ELSE
	nOutput := LIMIT(nMinValue, nTempOutput, nMaxValue);
	bEnableValveOutput := TRUE; 
END_IF

END_FUNCTION_BLOCK

// ---- Programs/P_Inputs.TcPOU
PROGRAM P_Inputs
VAR
	fbJoystick 				: FB_JoystickInputScaling;
	fbPositionSensor 		: FB_PositionInputScaling;
	fbPressureSupplySensor 	: FB_PressureInputScaling;
	fbPressureReturnSensor 	: FB_PressureInputScaling;
	fbPressurePistonSide 	: FB_PressureInputScaling;
	fbPressureLhvSide 		: FB_PressureInputScaling;
	fbPressureRodSide 		: FB_PressureInputScaling;
END_VAR

fbJoystick(
	bEnable := G_Inputs.bManualModeSelector,
	nRawInput := G_Inputs.stJoyY.nValue,
	fOutput => G_Sensors.fJoystickY
);

fbPositionSensor(
	nRawInput := G_Inputs.stCylPos.nValue,
	fOutput => G_Sensors.fPistonPosition
);

fbPressureSupplySensor(
	nRawInput := G_Inputs.stPressureSupply.nValue,
	fOutput => G_Sensors.fPressureSupply
);

fbPressureReturnSensor(
	nRawInput := G_Inputs.stPressureReturn.nValue,
	fOutput => G_Sensors.fPressureReturn
);

fbPressurePistonSide(
	nRawInput := G_Inputs.stPressurePistonSide.nValue,
	fOutput => G_Sensors.fPressurePistonSide
);

fbPressureLhvSide(
	nRawInput := G_Inputs.stPressureLhvSide.nValue,
	fOutput => G_Sensors.fPressureLhvSide
);

fbPressureRodSide(
	nRawInput := G_Inputs.stPressureRodSide.nValue,
	fOutput => G_Sensors.fPressureRodSide
);

END_PROGRAM

// ---- Inputs/FB_JoystickInputScaling.TcPOU
FUNCTION_BLOCK FB_JoystickInputScaling
VAR_INPUT
	bEnable : BOOL;
	nRawInput : INT;
END_VAR
VAR_OUTPUT
	fOutput : LREAL;
END_VAR
VAR
	fRawInput : LREAL;
	fTempInput : LREAL;
	fTempOutput : LREAL;
	fMaxInputValue			: LREAL := 14746.0;
	fMinInputValue 			: LREAL := 1617.0;
	fNeutralInputValue  	: LREAL := 8160.0;
	fNeutralDeadband		: LREAL := 50.0;
	fMaxOutputValue  		: LREAL := 1.0;
	fMinOutputValue  		: LREAL := -1.0;
	fNeutralOutputValue  	: LREAL := 0.0;
END_VAR

fRawInput := INT_TO_LREAL(nRawInput);

fTempInput := fRawInput - fNeutralInputValue;

IF fTempInput > fNeutralDeadband THEN
	fTempOutput := fTempInput/(fMaxInputValue - fNeutralInputValue);
ELSIF fTempInput < -fNeutralDeadband THEN	
	fTempOutput := fTempInput/(fNeutralInputValue - fMinInputValue);
ELSE
	fTempOutput := 0.0;
END_IF

IF NOT(bEnable) THEN
	fOutput := 0.0;
ELSE
	fOutput := LIMIT(fMinOutputValue, fTempOutput, fMaxOutputValue);
END_IF

END_FUNCTION_BLOCK

// ---- Inputs/FB_PositionInputScaling.TcPOU
FUNCTION_BLOCK FB_PositionInputScaling
VAR_INPUT
	nRawInput : INT;
END_VAR
VAR_OUTPUT
	fOutput : LREAL;
END_VAR
VAR
	fRawInput : LREAL;
	fNormalizedInput: LREAL;
	fMaxInputValue 			: LREAL := 16099.0;
	fMinInputValue			: LREAL := 125.0;
	fMaxOutputValue  		: LREAL := 0.5;
	fMinOutputValue  		: LREAL := 0.0;		
END_VAR

fRawInput := INT_TO_LREAL(nRawInput);

fNormalizedInput := (fRawInput - fMinInputValue) / (fMaxInputValue - fMinInputValue);

fOutput := LIMIT(fMinOutputValue, fMinOutputValue + fNormalizedInput*(fMaxOutputValue - fMinOutputValue), fMaxOutputValue);

END_FUNCTION_BLOCK

// ---- Inputs/FB_PressureInputScaling.TcPOU
FUNCTION_BLOCK FB_PressureInputScaling
VAR_INPUT
	nRawInput : INT;
END_VAR
VAR_OUTPUT
	fOutput : LREAL;
END_VAR
VAR
	fRawInput : LREAL;
	fNormalizedInput: LREAL;
	fMinInputValue			: LREAL := 0.0;
	fMaxInputValue			: LREAL := 32767.0;
	fMaxOutputValue 		: LREAL := 400.0;
	fMinOutputValue  		: LREAL := 0.0;			
END_VAR

fRawInput := INT_TO_LREAL(nRawInput);

fNormalizedInput := (fRawInput - fMinInputValue) / (fMaxInputValue - fMinInputValue);

fOutput := LIMIT(fMinOutputValue, fMinOutputValue + fNormalizedInput*(fMaxOutputValue - fMinOutputValue), fMaxOutputValue);

END_FUNCTION_BLOCK

// ---- Programs/P_Simulator.TcPOU
PROGRAM P_Simulator
VAR
	fbCraneSimulator : FB_CraneSimulator;
END_VAR

fbCraneSimulator(
	ssMethodType := BOOL_TO_SINT(G_Simulator.bSimulatorOn),
	uDCV := G_Work.fControlOutputNormalized,
	ppbar => G_Simulator.fPistonSidePressure,
	prbar => G_Simulator.fRodSidePressure,
	xm => G_Simulator.fPistonPosition
);

END_PROGRAM

// ---- GlobalTextList.TcGTLO
TEXTLIST GlobalTextList
  624 = '%0.1f'
  198 = '%f'
  949 = '%i'
  819 = '%s'
  850 = '%s '
  935 = '0.5m'
  892 = '0m'
  807 = '1m'
  948 = '1mx0'
  858 = 'Active Damping ON'
  175 = 'AUTO'
  885 = 'Automatic Control Settings'
  104 = 'Boom Angle: %0.1f [deg]'
  236 = 'Clock: %s [s]'
  920 = 'Closed Loop Position Control ON'
  214 = 'Comissioning'
  52 = 'ControlBox'
  109 = 'Controller Parameter Tuning'
  829 = 'Current I-gain: %0.1f '
  58 = 'Current Max Piston Stroke: %0.1f [m] '
  577 = 'Current MaxError: %0.1f '
  147 = 'Current MaxError: %0.1f [m] '
  196 = 'Current MaxError: %f [m] '
  955 = 'Current MaxFlow: %0.1f [L/min] '
  827 = 'Current MaxFlow: %0.1f [m] '
  137 = 'Current P-gain: %0.1f '
  668 = 'Current P-gain: %0.1f [m] '
  791 = 'Current Pgain: %0.1f [m] '
  907 = 'Current Position: %f [m] '
  471 = 'Cylinder Position Reference: %0.1f [m]'
  995 = 'Cylinder Position Reference: %f [m]'
  752 = 'Cylinder Velocity Reference: %0.0001f [m/s]'
  954 = 'Cylinder Velocity Reference: %0.01f [m/s]'
  105 = 'Cylinder Velocity Reference: %0.1f [m/s]'
  755 = 'Cylinder Velocity Reference: %0.1s [m/s]'
  25 = 'Cylinder Velocity Reference: %f [m/s]'
  308 = 'Cylinder Velocity Reference: %f [m]'
  30 = 'Cylinder Velocity Reference: %i'
  903 = 'Cylinder Velocity Reference: %s'
  128 = 'Cylinder Velocity Reference: %s [m/s]'
  556 = 'Down'
  501 = 'DOWN'
  353 = 'Enable'
  409 = 'ENABLE'
  527 = 'End Stop Status: %s '
  90 = 'FAULT'
  548 = 'Feed Forward Controller On'
  392 = 'Feed Forward Tuning'
  187 = 'Gain'
  904 = 'Hold Pos time: %0.1f [s] '
  445 = 'Integral Controller'
  81 = 'Integral Controller Gain'
  443 = 'Integral Controller On'
  573 = 'Integral Controller ON'
  961 = 'JOYSTICK Y'
  660 = 'MANUAL'
  8 = 'Manual Cylinder Position   Reference [m]'
  157 = 'Manual Cylinder Position Reference'
  11 = 'Manual Cylinder Position Reference [m]'
  7 = 'Max Piston Stroke: %0.1f [m] '
  110 = 'Max Piston Stroke: %f [m] '
  261 = 'Max Position Error'
  84 = 'Max Stroke: %f [m] '
  188 = 'Mode'
  76 = 'Mode: %s '
  415 = 'Motion Reference Generator Settings'
  655 = 'New I-gain: %0.1f '
  646 = 'New Max Piston Stroke: %0.1f [m] '
  895 = 'New MaxError: %0.1f '
  731 = 'New MaxError: %0.1f  [m]'
  683 = 'New MaxError: %f  [m]'
  330 = 'New MaxFlow: %0.1f [L/min] '
  993 = 'New MaxFlow: %0.1f [m] '
  347 = 'New P-gain: %0.1f '
  792 = 'New P-gain: %0.1f [m] '
  65 = 'OFF'
  629 = 'ON'
  751 = 'Pgain: %0.1f [m] '
  622 = 'Position SP: %0.1f [m] '
  463 = 'Position SP: %f [m] '
  651 = 'Proportional '
  705 = 'Proportional  Controller'
  982 = 'Proportional  Controller Gain'
  711 = 'Proportional Gain'
  215 = 'Ramp time: %0.1f [s] '
  310 = 'RUNNING'
  695 = 'Set New Value'
  466 = 'Simulation'
  279 = 'Start'
  868 = 'START'
  254 = 'START AUTO'
  149 = 'Start delay: %0.1f [m/s] '
  828 = 'Start delay: %0.1f [s] '
  324 = 'Start Position SP: %0.1f [m/s] '
  286 = 'Start Position: %0.1f [m] '
  78 = 'Start Position: %f [m] '
  253 = 'Start Velocity %0.1f [m/s] '
  314 = 'Start Velocity: %0.1f [m/s] '
  983 = 'Start Velocity: %f [m/s] '
  978 = 'Started'
  795 = 'Status'
  173 = 'Status: %s '
  397 = 'STOP'
  495 = 'Time: %0.1f [s]'
  221 = 'Time: %f [s]'
  61 = 'Time: %i [s]'
  725 = 'Time: %s [s]'
  932 = 'UP'
  638 = 'Velocity SP: %0.1f [m/s] '
  999 = 'Velocity SP: %f [m/s] '
  730 = 'VelocityFeed Forward Controller On'
  560 = 'VelocityFeed Forward Controller ON'
  444 = 'x0'
END_TEXTLIST

// ---- HMI/HMI.TcVIS
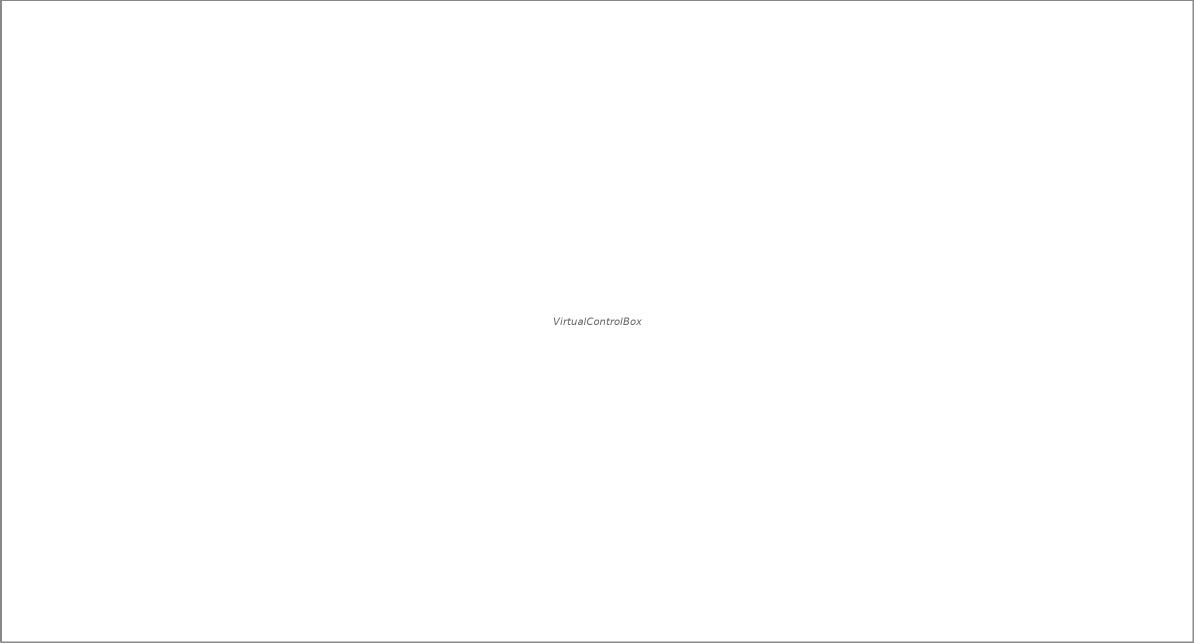
VISUALIZATION HMI  // 1194x643
    TabControl (1,0 1193x643)
        shows VirtualControlBox()
        shows CommissioningHMI()
        [0]: TabTitle=ControlBox
        [1]: TabTitle=Comissioning
END_VISUALIZATION

// ---- HMI/Sub/CommissioningHMI.TcVIS
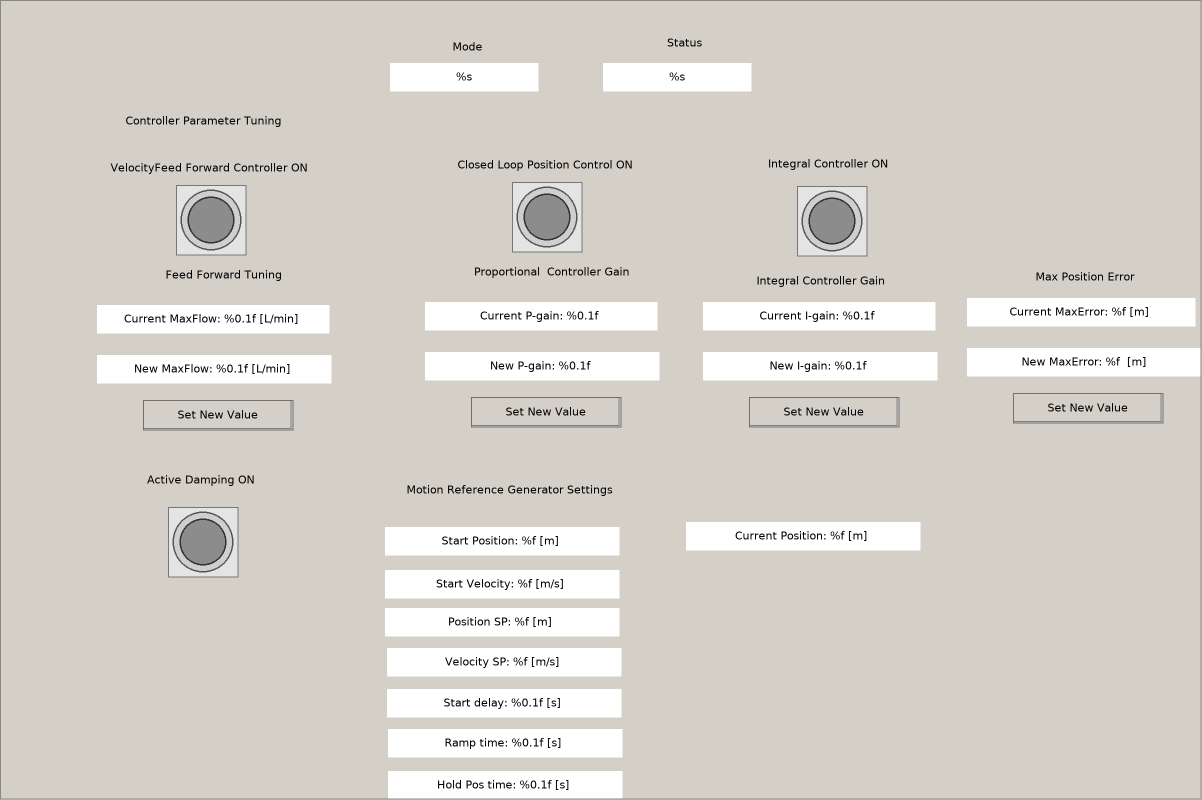
VISUALIZATION CommissioningHMI  // 1202x800
    Button (471,397 150x30), "Set New Value"
        tap G_Commissioning.bSetNewProportionalGain
    Textfield (424,301 234x30), "Current P-gain: %0.1f", text variable: G_Parameters.stParam.stClosedLoopControlSettings.fProportionalGain
    Textfield (424,351 236x30), "New P-gain: %0.1f", text variable: G_Commissioning.fNewProportionalGain
        OnMouseDown: write the text variable via Default
    Label (469,257 166x30), "Proportional Controller Gain"
    Button (749,397 150x30), "Set New Value"
        tap G_Commissioning.bSetNewIntegralGain
    Textfield (702,301 234x30), "Current I-gain: %0.1f", text variable: G_Parameters.stParam.stClosedLoopControlSettings.fIntegralGain
    Textfield (702,351 236x30), "New I-gain: %0.1f", text variable: G_Commissioning.fNewIntegralGain
        OnMouseDown: write the text variable via Default
    Label (746,266 150x30), "Integral Controller Gain"
    Label (94,106 219x30), "Controller Parameter Tuning"
    PushSwitch (797,186 70x70), variable: G_Commissioning.stAutomaticControlSettings.bEnableIntegralController, behaviour: TOGGLE, style: Switch-PushSwitch-Gray
    Label (745,149 166x30), "Integral Controller ON"
    Label (419,150 252x30), "Closed Loop Position Control ON"
    PushSwitch (512,182 70x70), variable: G_Commissioning.stAutomaticControlSettings.bEnableClosedLoopPositionControl, behaviour: TOGGLE, style: Switch-PushSwitch-Gray
    Label (83,153 252x30), "VelocityFeed Forward Controller ON"
    PushSwitch (176,185 70x70), variable: G_Commissioning.stAutomaticControlSettings.bEnableVelocityFeedForwardControl, behaviour: TOGGLE, style: Switch-PushSwitch-Gray
    PushSwitch (168,507 70x70), variable: G_Commissioning.stAutomaticControlSettings.bEnableActiveDamping, behaviour: TOGGLE, style: Switch-PushSwitch-Gray
    Label (75,465 252x30), "Active Damping ON"
    Button (143,400 150x30), "Set New Value"
        tap G_Commissioning.bSetNewMaxFlowCapacity
    Textfield (96,304 234x30), "Current MaxFlow: %0.1f [L/min]", text variable: G_Parameters.stParam.stOpenLoopControlSettings.fMaxFlowCapacity
    Textfield (96,354 236x30), "New MaxFlow: %0.1f [L/min]", text variable: G_Commissioning.fNewMaxFlowCapacity
        OnMouseDown: write the text variable via Default, min 0, max 40
    Label (141,260 166x30), "Feed Forward Tuning"
    Button (1013,393 150x30), "Set New Value"
        tap G_Commissioning.bSetNewMaxPositionError
    Textfield (966,297 230x30), "Current MaxError: %f [m]", text variable: G_Parameters.stParam.stClosedLoopControlSettings.fMaxPositionError
    Textfield (966,347 236x30), "New MaxError: %f [m]", text variable: G_Commissioning.fNewMaxPositionError
        OnMouseDown: write the text variable via Default
    Label (1010,262 150x30), "Max Position Error"
    Label (412,32 111x30), "Mode"
    Label (629,28 111x30), "Status"
    Textfield (389,62 150x30), "%s", text variable: G_Work.eMode
    Textfield (602,62 150x30), "%s", text variable: G_Work.eStatus
    Label (364,475 291x30), "Motion Reference Generator Settings"
    Textfield (384,526 236x30), "Start Position: %f [m]", text variable: G_Commissioning.stMotionReferenceGeneratorSettings.fStartPosition_m
        OnMouseDown: write the text variable via Default, min 0, max 0.5
    Textfield (384,569 236x30), "Start Velocity: %f [m/s]", text variable: G_Commissioning.stMotionReferenceGeneratorSettings.fStartVelocity_m
        OnMouseDown: write the text variable via Default, min 0, max 0.05
    Textfield (384,607 236x30), "Position SP: %f [m]", text variable: G_Commissioning.stMotionReferenceGeneratorSettings.fPositionSetpoint_ms
        OnMouseDown: write the text variable via Default, min 0, max 0.45
    Textfield (386,647 236x30), "Velocity SP: %f [m/s]", text variable: G_Commissioning.stMotionReferenceGeneratorSettings.fVelocitySetpoint_m
        OnMouseDown: write the text variable via Default, min 0, max 0.05
    Textfield (386,688 236x30), "Start delay: %0.1f [s]", text variable: G_Commissioning.stMotionReferenceGeneratorSettings.fTimeBeforeStarting_s
        OnMouseDown: write the text variable via Default, min 0, max 10
    Textfield (387,728 236x30), "Ramp time: %0.1f [s]", text variable: G_Commissioning.stMotionReferenceGeneratorSettings.fRampTime_s
        OnMouseDown: write the text variable via Default, min 0, max 10
    Textfield (387,770 236x30), "Hold Pos time: %0.1f [s]", text variable: G_Commissioning.stMotionReferenceGeneratorSettings.fHoldPositionTime_s
        OnMouseDown: write the text variable via Default, min 0, max 10
    Textfield (685,521 236x30), "Current Position: %f [m]", text variable: G_Sensors.fPistonPosition
        OnMouseDown: write the text variable via Default, min 0, max 0.5
END_VISUALIZATION

// ---- HMI/Sub/VirtualControlBox.TcVIS
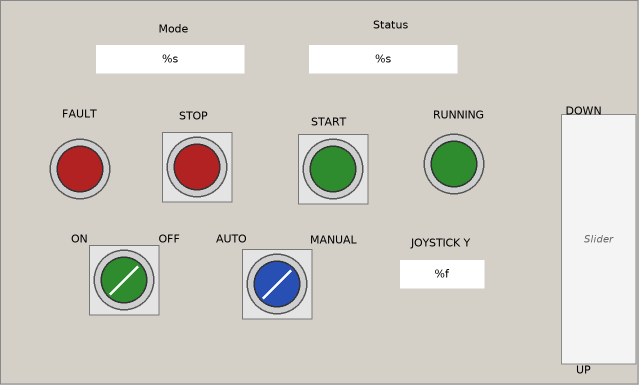
VISUALIZATION VirtualControlBox  // 639x385
    Lamp1 (419,129 70x70), variable: G_VirtualControlBox.bGreenLight, style: Lamp-Lamp1-Green
    Lamp1 (45,134 70x70), variable: G_VirtualControlBox.bRedLight, style: Lamp-Lamp1-Red
    PushSwitch (162,132 70x70), variable: G_VirtualControlBox.bStopButton, behaviour: TAP, style: Switch-PushSwitch-Red
    PushSwitch (298,134 70x70), variable: G_VirtualControlBox.bStartButton, behaviour: TAP, style: Switch-PushSwitch-Green
    RotarySwitch (89,245 70x70), variable: G_VirtualControlBox.bOnSelector, behaviour: TOGGLE, style: Switch-RotarySwitch-Green
    Label (51,224 57x30), "ON"
    Label (141,224 57x30), "OFF"
    RotarySwitch (242,249 70x70), variable: G_VirtualControlBox.bAutoSelector, behaviour: TOGGLE, style: Switch-RotarySwitch-Blue
    Label (203,224 57x30), "AUTO"
    Label (305,225 57x30), "MANUAL"
    Slider (561,114 75x250), variable: G_VirtualControlBox.fJoystickY, scale -1..1
    Label (51,99 57x30), "FAULT"
    Label (430,100 57x30), "RUNNING"
    Label (300,107 57x30), "START"
    Label (165,101 57x30), "STOP"
    Label (385,228 111x30), "JOYSTICK Y"
    Textfield (399,259 86x30), "%f", text variable: G_VirtualControlBox.fJoystickY
        OnMouseClick: write the text variable via Default, min -1, max 1
    Label (118,14 111x30), "Mode"
    Label (335,10 111x30), "Status"
    Textfield (95,44 150x30), "%s", text variable: G_Work.eMode
    Textfield (308,44 150x30), "%s", text variable: G_Work.eStatus
    Label (528,96 111x30), "DOWN"
    Label (528,355 111x30), "UP"
END_VISUALIZATION
